{region '#Template'}
	{attribute 'Version' := '1.2.1.0'}
	{attribute 'Tags' := '"LCID": "1031", "Text": "General, Cabinet, Control cabinet"'}
	{attribute 'Tags' := '"LCID": "1033", "Text": "General, Cabinet, Control cabinet"'}
	{attribute 'Using' := '"Type": "Template", "URI": "EC_AMEV"'}
	{attribute 'Description' := '"LCID": "1031", "Text": "Schaltschrank Ereignisse"'}
	{attribute 'Description' := '"LCID": "1033", "Text": "Control cabinet events"'}
{endregion}
FUNCTION_BLOCK FB_BA_ControlCabinet EXTENDS FB_BA_ControlCabinetBasic
VAR_INPUT CONSTANT
	Fuse01					: FB_BA_SensorBinary_IO;		
	Fuse02					: FB_BA_SensorBinary_IO;	
	Fuse03					: FB_BA_SensorBinary_IO;	
END_VAR

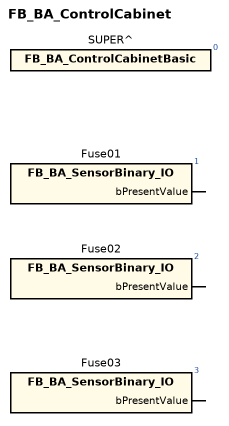
SUPER^(); // FB_BA_ControlCabinetBasic
Fuse01(); // FB_BA_SensorBinary_IO
Fuse02(); // FB_BA_SensorBinary_IO
Fuse03(); // FB_BA_SensorBinary_IO

METHOD FB_init : BOOL
VAR_INPUT
	bInitRetains : BOOL; // if TRUE, the retain variables are initialized (warm start / cold start)
	bInCopyCode : BOOL;  // if TRUE, the instance afterwards gets moved into the copy code (online change)
END_VAR
Fuse01.iParent								:= THIS^;		
Fuse01.iLabel 								:= LblCmpGeneral.ControlCabinet_Fuse;	
Fuse01.sObjectName							:= '{Idx=01}';
Fuse01.eDPADMode							:= E_BA_DPADMode.eInclude;																						
Fuse01.Input.iLabel							:= LblCmpGeneral.ControlCabinet_Fuse_Input;	
Fuse01.Input.sObjectName					:= '{Idx=01}';	
Fuse01.Input.ePolarity						:= E_BA_Polarity.eReverse;
Fuse01.Input.sActiveText 					:= txtEvent_Triggered;
Fuse01.Input.sInactiveText 					:= txtEvent_Normal;
Fuse01.Input.nEventClassID					:= EC_ID.NC30;
Fuse01.Input.aEventTransitionText[1]		:= txtEvent_Triggered;
Fuse01.Input.aEventTransitionText[2]		:= txtEvent_Error;
Fuse01.Input.aEventTransitionText[3]		:= txtEvent_Normal;
Fuse01.Input.bEventDetectionEnable			:= TRUE;
Fuse01.Input.aEventEnable[1]				:= TRUE;			//	to_offnormal
Fuse01.Input.aEventEnable[2]				:= TRUE;			//	to_fault
Fuse01.Input.aEventEnable[3]				:= TRUE;			//	to_normal
Fuse01.Input.eEnPlantLock					:= E_BA_LockPriority.eNoLock;	
								 
Fuse02.iParent								:= THIS^;		
Fuse02.iLabel 								:= LblCmpGeneral.ControlCabinet_Fuse;	
Fuse02.sObjectName							:= '{Idx=02}';
Fuse02.eDPADMode							:= E_BA_DPADMode.eInclude;																						
Fuse02.Input.iLabel							:= LblCmpGeneral.ControlCabinet_Fuse_Input;	
Fuse02.Input.sObjectName					:= '{Idx=02}';	
Fuse02.Input.ePolarity						:= E_BA_Polarity.eReverse;
Fuse02.Input.sActiveText 					:= txtEvent_Triggered;
Fuse02.Input.sInactiveText 					:= txtEvent_Normal;
Fuse02.Input.nEventClassID					:= EC_ID.NC30;
Fuse02.Input.aEventTransitionText[2]		:= txtEvent_Error;
Fuse02.Input.aEventTransitionText[3]		:= txtEvent_Normal;
Fuse02.Input.bEventDetectionEnable			:= TRUE;
Fuse02.Input.aEventEnable[1]				:= TRUE;			//	to_offnormal
Fuse02.Input.aEventEnable[2]				:= TRUE;			//	to_fault
Fuse02.Input.aEventEnable[3]				:= TRUE;			//	to_normal
Fuse02.Input.eEnPlantLock					:= E_BA_LockPriority.eNoLock;	
										 
Fuse03.iParent								:= THIS^;		
Fuse03.iLabel 								:= LblCmpGeneral.ControlCabinet_Fuse;	
Fuse03.sObjectName							:= '{Idx=03}';
Fuse03.eDPADMode							:= E_BA_DPADMode.eInclude;																						
Fuse03.Input.iLabel							:= LblCmpGeneral.ControlCabinet_Fuse_Input;	
Fuse03.Input.sObjectName					:= '{Idx=03}';	
Fuse03.Input.ePolarity						:= E_BA_Polarity.eReverse;
Fuse03.Input.sActiveText 					:= txtEvent_Triggered;
Fuse03.Input.sInactiveText 					:= txtEvent_Normal;
Fuse03.Input.nEventClassID					:= EC_ID.NC30;
Fuse03.Input.aEventTransitionText[1]		:= txtEvent_Triggered;
Fuse03.Input.aEventTransitionText[2]		:= txtEvent_Error;
Fuse03.Input.aEventTransitionText[3]		:= txtEvent_Normal;
Fuse03.Input.bEventDetectionEnable			:= TRUE;
Fuse03.Input.aEventEnable[1]				:= TRUE;			//	to_offnormal
Fuse03.Input.aEventEnable[2]				:= TRUE;			//	to_fault
Fuse03.Input.aEventEnable[3]				:= TRUE;			//	to_normal
Fuse03.Input.eEnPlantLock					:= E_BA_LockPriority.eNoLock;
END_METHOD

END_FUNCTION_BLOCK

(* stored: Version 1.1.0.1, ProductVersion 3.1.4024.9
   POU FB_BA_ControlCabinet: Id {590e0131-10bc-49bc-b8fd-be0c20d77b39}, SpecialFunc None
   Method FB_init: Id {9094676e-9e13-4c8b-baeb-e793e496ccfc} *)
